FUNCTION_BLOCK AX_TONOF (* standard timer function block (on/off-delay timing) *)
  (* Standard: 61499-2; Classification: standard timer function block; Description: Copyright (c) 2024 HR Agrartechnik GmbH This program and the accompanying materials are made available under the terms of the Eclipse Public License 2.0 which is available at https://www.eclipse.org/legal/epl-2.0/ SPDX-License-Identifier: EPL-2.0 *)
  (* Version 3.0, 2025-04-14, Patrick Aigner, changed package *)
  (* Version 1.1, 2024-04-23, Franz Hoepfinger, HR Agrartechnik GmbH, Add a Reset to Timer FBs *)
  (* Version 1.0, 2024-03-04, Franz Hoepfinger, HR Agrartechnik GmbH *)
  PACKAGE adapter::events::unidirectional::timers;
  IMPORT eclipse4diac::core::TypeHash;
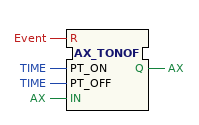
  EVENT_INPUT
    R; (* Reset *)
  END_EVENT
  VAR_INPUT
    PT_ON : TIME; (* Process time ON Delay *)
    PT_OFF : TIME; (* Process time OFF Delay *)
  END_VAR
  SOCKETS
    IN : adapter::types::unidirectional::AX; (* Input *)
  END_SOCKETS
  PLUGS
    Q : adapter::types::unidirectional::AX; (* Output *)
  END_PLUGS
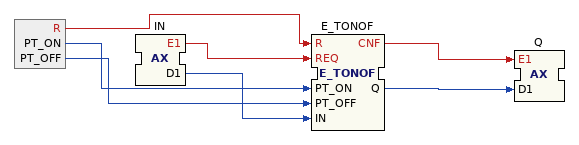
  FBS
    E_TONOF : iec61499::events::timers::E_TONOF;
  END_FBS
  EVENT_CONNECTIONS
    R TO E_TONOF.R;
    IN.E1 TO E_TONOF.REQ;
    E_TONOF.CNF TO Q.E1;
  END_CONNECTIONS
  DATA_CONNECTIONS
    PT_ON TO E_TONOF.PT_ON;
    PT_OFF TO E_TONOF.PT_OFF;
    IN.D1 TO E_TONOF.IN;
    E_TONOF.Q TO Q.D1;
  END_CONNECTIONS
END_FUNCTION_BLOCK
